PROGRAM PumpDownProgramm
VAR

END_VAR

(*Kompressor wird angeschaltet*)	
	KP_ON		:= TRUE;	
	PID_KP.Aktiv:= TRUE;
		
(*Schütze, EV werden für PumpDown Modus geschaltet*)
 	IF bPumpDown THEN 	
	bPumpDown_rev := FALSE;
	fb_Schuetzstellung(myStatus:= PumpDown);
	
	(*Pump-Down wird durchgeführt bis der Druck vor dem KP kleiner als 1,4 Bar ist*)	
		IF   PT_VD_out.rDruck < Soll_PumpDownDruck THEN  			//!!Ist noch nicht ansprechbar!!
			bPumpDown := FALSE;
			bPumpDownAbgeschlossen:= TRUE;
			
			(*Kompressor wird ausgeschaltet*)	
			KP_ON		:= FALSE;	
			PID_KP.Aktiv:= FALSE;
		END_IF
	END_IF

(*Schütze, EV_rev werden für PumpDown_rev Modus geschaltet*)
	IF bPumpDown_rev THEN 
	bPumpDown := FALSE;	
	fb_Schuetzstellung(myStatus:= PumpDown_rev);
	
	(*Pump-Down wird durchgeführt bis der Druck vor dem KP kleiner als 1,4 Bar ist*)	
		IF  PT_KP_out.rDruck < Soll_PumpDownDruck THEN  			//!!Ist noch nicht ansprechbar!!
			bPumpDown_rev := FALSE;
			bPumpDown_revAbgeschlossen:= TRUE;
			
			(*Kompressor wird ausgeschaltet*)	
			KP_ON		:= FALSE;	
			PID_KP.Aktiv:= FALSE;
		END_IF
	END_IF

END_PROGRAM

(* stored: Version 1.1.0.1, ProductVersion 3.1.4019.2
   POU PumpDownProgramm: Id {6f105f69-9598-4667-a3f9-d4c4a9e74e4d}, SpecialFunc None *)
